VAR_GLOBAL

Axis1	:	AXIS_REF;
Axis2	:	AXIS_REF;


END_VAR

(* stored: Version 1.1.0.1, ProductVersion 3.1.4022.18
   GVL GVL_Motion: Id {3ce66b51-07dc-4637-8223-34f1ff34f6e2} *)
